PROGRAM prgVoiceSynsthesis
VAR
END_VAR

END_PROGRAM

(* stored: Version 1.1.0.1, ProductVersion 3.1.4024.3
   POU prgVoiceSynsthesis: Id {292cc062-60d1-4444-bd9b-a3719ebf2528}, SpecialFunc None *)
